Universal Robots PolyScope program: p2_Group1_v1.urp

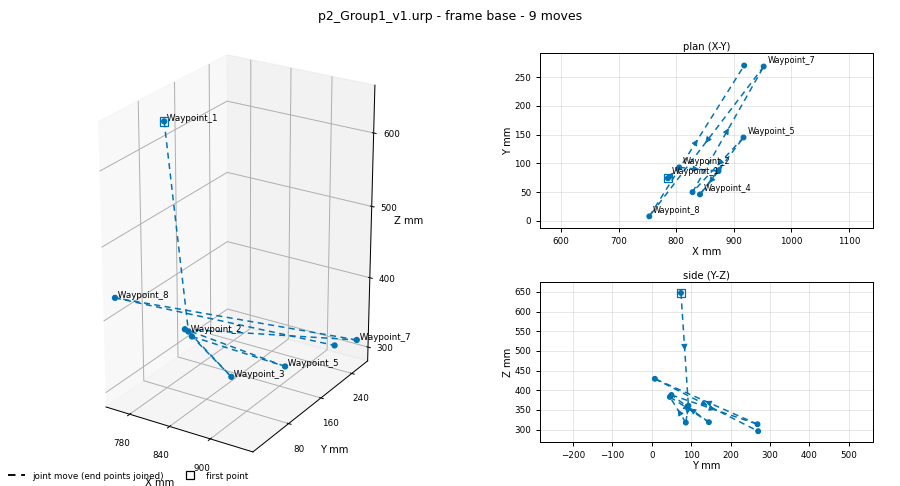
[picture p0: tool path of p2_Group1_v1.urp in frame base, 9 of 9 moves have a stored position in this frame; points joined in program order, loops and branches not executed]
Program p2_Group1_v1 (installation=default directory=/programs/usbdisk/Project 2_v1 createdIn=5.13.0 lastSavedIn=5.13.0 robotSerialNumber=20225201357)
Calibrated DH parameters: a=[-0.000097, -0.065329, -0.560646, 0.000001, -0.00004, 0]; d=[0.180831, -263.113709, 285.24385, -21.955837, 0.119737, 0.115719]; alpha=[1.571643, -0.002312, 0.004975, 1.569542, -1.570894, 0]; deltaTheta=[0, 1.463798, 5.013296, -0.193909, 0, 0]
InitVariablesNode
Robot Program (runOnlyOnce=false)
  robotState := read_port_register(200)
  If robotState≟0
    MoveJ speed 60 deg/s, acceleration 80 deg/s^2 (useActiveTCP=true) feature=Base
      Waypoint Waypoint_1: motionParameters(nextMotionTime=3); TCP in base x=785.448 y=74.147 z=647.122 mm, rx=-0.5336 ry=-1.0414 rz=0.0693 rad; joints [43.681, -78.245, -124.259, 12.74, 31.722, 71.465] deg; TCP offset x=-0.19 y=3.58 z=256.26 mm, rx=0.0015 ry=-2.7841 rz=0 rad
      Waypoint Waypoint_2: TCP in base x=805.005 y=93.045 z=360.866 mm, rx=-0.2336 ry=-0.9663 rz=-0.1947 rad; joints [43.676, -96.332, -136.356, 27.356, 31.716, 105.556] deg
      Waypoint Waypoint_3: motionParameters(nextMotionTime=3); TCP in base x=873.289 y=86.447 z=318.022 mm, rx=-0.5459 ry=-1.0606 rz=-0.6071 rad; joints [44.07, -112.542, -122.005, -8.87, 3.116, 146.418] deg
  ElseIf robotState≟1
    MoveJ speed 60 deg/s, acceleration 80 deg/s^2 (useActiveTCP=true) feature=Base
      Waypoint Waypoint_4: motionParameters(nextMotionTime=1); TCP in base x=841.207 y=46.002 z=383.12 mm, rx=-0.9277 ry=-1.0657 rz=-0.5165 rad; joints [43.103, -112.546, -122.88, -8.862, -9.396, 130.779] deg
      Waypoint Waypoint_5: motionParameters(nextMotionTime=1); TCP in base x=916.899 y=145.053 z=319.05 mm, rx=-0.7729 ry=-0.8712 rz=-0.3486 rad; joints [44.815, -113.524, -115.202, -19.553, 6.421, 130.441] deg
      Waypoint Waypoint_6: motionParameters(nextMotionTime=1); TCP in base x=828.231 y=49.963 z=388.09 mm, rx=-1.0777 ry=-1.0794 rz=-0.455 rad; joints [43.495, -113.49, -124.38, -13.278, -14.927, 130.818] deg
      Waypoint Waypoint_7: motionParameters(nextMotionTime=0.5); TCP in base x=951.995 y=268.396 z=313.832 mm, rx=-0.0597 ry=-0.8617 rz=-0.37 rad; joints [44.955, -110.895, -113.802, 4.881, 33.475, 130.807] deg
      Waypoint Waypoint_8: motionParameters(nextMotionTime=0.5); TCP in base x=753.101 y=7.857 z=429.233 mm, rx=-0.907 ry=-1.2385 rz=-0.6808 rad; joints [44.904, -110.887, -128.86, 4.902, -19.188, 130.847] deg
      Waypoint Waypoint_9: motionParameters(nextMotionTime=0.5); TCP in base x=918.087 y=270.137 z=296.16 mm, rx=-0.1426 ry=-0.8789 rz=-0.3478 rad; joints [47.877, -110.885, -117.165, 4.898, 28.437, 130.73] deg
